// TIA Portal V20 export
TYPE "LER_typeStatusReelcut"
// stored: Access Published
   STRUCT
      anodeReelcutStart : Bool;
      anodeReelcutRunCheck : Bool;
      cathodeReelcutStart : Bool;
      cathodeReelcutRunCheck : Bool;
      stackStop : Bool;
      stackStopCheck : Bool;
      forceStop : Bool;
      forceStopComplete : Bool;
      anodeSize : LReal;
      anodeReelcutPrePosition : LReal;
      anodeReelcutCount : LReal;
      anodeReelcutVelocity : LReal;
      anodeReelcutAcceleration : LReal;
      anodeReelcutDeceleration : LReal;
      anodeStart_anodeRunOffset : LReal;
      anodeStart_cathodeRunOffset : LReal;
      anodeStart_anodeRunTimeOffset : LReal;
      anodeStart_cathodeRunTimeOffset : LReal;
      cathodeSize : LReal;
      cathodeReelcutPrePosition : LReal;
      cathodeReelcutCount : LReal;
      cathodeReelcutVelocity : LReal;
      cathodeReelcutAcceleration : LReal;
      cathodeReelcutDeceleration : LReal;
      cathodeStart_anodeRunOffset : LReal;
      cathodeStart_cathodeRunOffset : LReal;
      cathodeStart_anodeRunTimeOffset : LReal;
      cathodeStart_cathodeRunTimeOffset : LReal;
   END_STRUCT;
END_TYPE
